{attribute 'qualified_only'}
{attribute 'strict'}
TYPE E_MessageNumbers :
(
	// no messages
		NA_NoMessage		:= 0, // no message active
	// System faults
		FF_Unknown 			:= 1, // unknown error occured 
		FF_NoCommunication 	:= 2, // no communication detected
		FF_ComunicationFault:= 3, // Communication error detected (does not match expected com)
		FF_Overload			:= 4, // hardware overload detected
		FF_EncoderFault		:= 5, // encoder signal incorrect or not present
		FF_SlaveFault		:= 6, // slave system is has active fatal fault
		FF_AxisFault		:= 7, // Axis fault feedback
		FF_DriveFault		:= 8, // Axis drive fault
		FF_Collision		:= 9, // Collision detected between 2 or more parts of the machine
	// Hardware faults
		CF_FeedbackFault		:= 100,	// Hardware feedback is does not match expected
		CF_WrongDirection		:= 101, // Hardware moving in incorrect direction
		CF_MoveToFast			:= 102, // Hardware movement completion time is lower then minimum
		CF_MoveToSlow			:= 103, // hardware movement maximum time was exceeded
		CF_WrongPosition		:= 104,	// Hardware is at different position then expected
		CF_Obstruction			:= 105, // Obstruction detected in movement path
	// Missing conditions
		MC_WaitingForproduct	:= 200,	// Waiting for product
		MC_WaitingForOperator	:= 201, // Waiting for operator action
		MC_WaitingForModule		:= 202,	// Waiting for other module
		MC_WaitingForMaster		:= 203, // Waiting Waiting for master
		MC_WaitingForSlave		:= 204, // waiting for slave
		MC_WrongPosition		:= 205, // Action or command not possible in current position
	// Operator messages
		OM_AlmostEmpty			:= 300, // product is almost empty refil is required
		OM_Finished 			:= 301, // product or action is finished
		OM_ready				:= 302, // ready for new task
	// Test Messages
		FF_MessageTest			:= 900, // Fatal fault message test
		CF_MessageTest			:= 901, // Cycle fault message test
		MC_MessageTest			:= 902, // Missing condition message test
		OM_MessageTest			:= 903	// Operator message test
)UDINT;
END_TYPE

(* stored: Version 1.1.0.1, ProductVersion 3.1.4024.3
   EnumerationTextList E_MessageNumbers: Id {d5d66a3f-bc78-479d-b404-0f4065b4a891} *)
